TYPE VARTYPE_EXTCANQUEUE:
STRUCT
	length: UINT;
	cobId: UDINT;
	rxData: ARRAY [0..7] OF USINT;
END_STRUCT
END_TYPE

(* stored: Version 1.1.0.1, ProductVersion 3.1.4024.9
   DUT VARTYPE_EXTCANQUEUE: Id {51215c44-60a8-4eeb-90e6-01936e0863cd} *)
